// TIA Portal V20 export
DATA_BLOCK "BA010AZCRRF1_AntennaLeft"   // DB3
AUTHOR : SIMATIC
FAMILY : Ident
VERSION : 1.2
// stored: InstanceOfName TO_IDENT, OfSystemLibElement TO_IDENT, OfSystemLibVersion 1.2
TO_IDENT   // technology object, version 1.2
   // VAR
   //    HW_ID { ExternalWritable := 'False'; S7_SetPoint := 'True'} : Word := 16#0249;
   //    CM_CHANNEL { ExternalWritable := 'False'; S7_SetPoint := 'True'} : Int := 1;
   //    LADDR { ExternalWritable := 'False'; S7_SetPoint := 'True'} : Word := 16#2AF8;
   //    CONFIGURATION { S7_SetPoint := 'True'} : IID_IN_PARAMETERS;
   //    DIAGNOSTIC { ExternalWritable := 'False'; S7_SetPoint := 'True'} : IID_IN_DIAGNOSTIC;
   //    STATIC { ExternalWritable := 'False'; S7_SetPoint := 'True'} : IID_IN_SYNC_TO;
   // END_VAR
BEGIN
   CONFIGURATION.config_mode := 16#01;
   CONFIGURATION.connected_reader := 16#0000;
   CONFIGURATION.param_buffer[1..16] := 16#00;
   STATIC.auto_reset_enabled := TRUE;
END_DATA_BLOCK
